INTERFACE I_Metadata EXTENDS I_Disposable, I_Serializable

METHOD PUBLIC Accept
VAR_INPUT
	Visitor : I_MetadataVisitor;
END_VAR
END_METHOD

PROPERTY PUBLIC Data : I_DataType
GET
END_GET
END_PROPERTY

PROPERTY PUBLIC Name : T_MAXSTRING
GET
END_GET
END_PROPERTY

METHOD PUBLIC SerializeWith
VAR_INPUT
	Serializer : I_Serializer;
END_VAR
END_METHOD

END_INTERFACE

(* stored: Version 1.1.0.1, ProductVersion 3.1.4024.12
   Itf I_Metadata: Id {b3ff1f0d-66e5-4d74-bc1c-93275596b47e}
   Method Accept: Id {b40cc3f0-b84a-4d50-8d80-6038db1973b9}
   Property Data: Id {b7855313-3f6b-071a-2940-a3c23cc0c517}
   Get Get: Id {4d6ad305-0619-0bdc-24bc-1943e07717f7}
   Property Name: Id {a976b692-b413-4da8-8139-60908d7dd759}
   Get Get: Id {4593a570-1b6e-4626-aead-cc492a933f45}
   Method SerializeWith: Id {a9e244ba-5227-41f1-a6d5-b2b58d6d0ec1} *)
